// TIA Portal V19 export
DATA_BLOCK "InstMainFB"   // DB10
TITLE = InstMainFB
{ DB_Accessible_From_OPC_UA := 'FALSE' }
// IDB MainFB
// stored: AssignedProDiagFB LiftProDiagFB, DBAccessibleFromOPCUA false, InstanceOfName MainFB, InstanceOfType FB
"MainFB"
   // VAR_INPUT
   //    Initial_Call { ExternalAccessible := 'False'; ExternalVisible := 'False'; ExternalWritable := 'False'} : Bool;
   // END_VAR
   // VAR
   //    instCommon { ExternalAccessible := 'False'; ExternalVisible := 'False'; ExternalWritable := 'False'; S7_SetPoint := 'True'} : "Common";
   //    instLift1Cmd { ExternalAccessible := 'False'; ExternalVisible := 'False'; ExternalWritable := 'False'; S7_SetPoint := 'True'} : "LiftCmd";
   //    instLift2Cmd { ExternalAccessible := 'False'; ExternalVisible := 'False'; ExternalWritable := 'False'; S7_SetPoint := 'True'} : "LiftCmd";
   //    instLiftSim { ExternalAccessible := 'False'; ExternalVisible := 'False'; ExternalWritable := 'False'; S7_SetPoint := 'True'} : "LiftSim";
   // END_VAR
BEGIN
END_DATA_BLOCK
